FUNCTION_BLOCK ABSTRACT FB_StateSpaceModel
VAR
    nx : INT;
    nu : INT;
    ny : INT;
	
    x  		: ARRAY[1..15] OF LREAL;

    _A  : ARRAY[1..15,1..15] OF LREAL;
    _B  : ARRAY[1..15,1..15] OF LREAL;
    _C  : ARRAY[1..15,1..15] OF LREAL;
    _D  : ARRAY[1..15,1..15] OF LREAL;
    _K  : ARRAY[1..15] OF LREAL;

	_activateObserver : BOOL;
    bInit : BOOL;
	
	i,j : INT;
    x_new : ARRAY[1..10] OF LREAL;
    e : LREAL;
END_VAR
VAR_OUTPUT
	y  : ARRAY[1..15] OF LREAL;
END_VAR

METHOD PUBLIC Init
VAR_INPUT
	activateObserver : BOOL;
END_VAR
VAR
    i,j : INT;
END_VAR

FOR i := 1 TO nx DO
    x[i] := 0;
    _K[i] := _K[i]; // keep
END_FOR
_activateObserver := activateObserver;
bInit := TRUE;
END_METHOD

METHOD PUBLIC Step
VAR_INPUT
    u  		: ARRAY[1..15] OF LREAL;
	y_meas 	: LREAL;
END_VAR

// --- Output ---
FOR i := 1 TO ny DO
    y[i] := 0;
    FOR j := 1 TO nx DO 
        y[i] := y[i] + _C[i,j]*x[j];
    END_FOR
END_FOR

// --- Innovation (single y example) ---
IF _activateObserver THEN
	e := y_meas - y[1];
ELSE 
	e := 0;
END_IF

// --- State update ---
FOR i := 1 TO nx DO
    x_new[i] := 0;

    FOR j := 1 TO nx DO
        x_new[i] := x_new[i] + _A[i,j]*x[j];
    END_FOR

    FOR j := 1 TO nu DO
        x_new[i] := x_new[i] + _B[i,j]*u[j];
    END_FOR

    x_new[i] := x_new[i] + _K[i]*e;
END_FOR

FOR i := 1 TO nx DO
    x[i] := x_new[i];
END_FOR
END_METHOD

END_FUNCTION_BLOCK

(* stored: Version 1.1.0.1, ProductVersion 3.1.4024.9
   POU FB_StateSpaceModel: Id {dcf04b36-9606-4b0e-bcf8-fd602d1b7f4c}, SpecialFunc None
   Method Init: Id {b1a1fbce-7488-459e-a918-05d26a30116b}
   Method step: Id {673a3b0c-a3cb-4aba-bf8c-343c4d6c442b} *)
